(* IEC 61131-3 sources: programs/VI-54/VI-54_20171205/VI-54_20171205/Stations/PLC_VI54/VI-54_171014/Class/Recipe_Camera, 1 file *)

(* ---- Recipe_Camera.st ---- *)
(*!
<Class
	Name               = "Recipe_Camera"
	Revision           = "0.0"
	RealtimeTask       = "false"
	CyclicTask         = "false"
	BackgroundTask     = "false"
	Sigmatek           = "false"
	OSInterface        = "false"
	HighPriority       = "false"
	Automatic          = "false"
	UpdateMode         = "Prescan"
	SharedCommandTable = "true"
	Objectsize         = "(810,120)">
	<Channels>
		<Server Name="TriggerOffset" Visualized="true" Initialize="false" WriteProtected="false" Retentive="false"/>
	</Channels>
	<Separators>
		<Servers>
			<SepChn Position="0"/>
		</Servers>
	</Separators>
	<Network Name="Recipe_Camera">
		<!-- List of Components in this network -->
		<Components>
			<Object
				Name       = "_base"
				Class      = "RecipeBase"
				Position   = "(218,120)"
				Visualized = "false">
				<Channels>
					<Server Name="Comm"/>
					<Client Name="MainRecipe"/>
				</Channels>
			</Object>
		</Components>
		<Comments>
		</Comments>
		<!-- List of Connections in this network -->
		<Connections>
			<Connection Source="this.Comm" Destination="_base.Comm" Vertices="(690,210),(518,210),"/>
			<Connection Source="_base.MainRecipe" Destination="this.MainRecipe" Vertices="(218,210),(38,210),"/>
		</Connections>
		<!-- Headerfiles -->
		<Options>
		</Options>
	</Network>
</Class>
*)
#pragma using RecipeBase

Recipe_Camera : CLASS
: RecipeBase
  //Servers:
	TriggerOffset 	: SvrCh_DINT;
  //Clients:
  //Variables:
  //Functions:

	FUNCTION VIRTUAL GLOBAL TriggerOffset::Write
		VAR_INPUT
			input (EAX) 	: DINT;
		END_VAR
		VAR_OUTPUT
			result (EAX) 	: DINT;
		END_VAR;
  //Tables:
	FUNCTION @STD
		VAR_OUTPUT
			ret_code	: CONFSTATES;
		END_VAR;
	FUNCTION GLOBAL TAB @CT_;
END_CLASS;

FUNCTION VIRTUAL GLOBAL Recipe_Camera::TriggerOffset::Write
	VAR_INPUT
		input (EAX) 	: DINT;
	END_VAR
	VAR_OUTPUT
		result (EAX) 	: DINT;
	END_VAR

	TriggerOffset := input;
  ReceptPtr^.Camera.TriggerOffset := TriggerOffset;
	result := TriggerOffset;

END_FUNCTION
